TYPE ST_FastDoorStates :
STRUCT
	eState		: E_FastDoorState; //State
	eLastState	: E_FastDoorState; //Last state
END_STRUCT
END_TYPE

(* stored: Version 1.1.0.1, ProductVersion 3.1.4024.9
   DUT ST_FastDoorStates: Id {4c93962d-641b-476f-b7dc-0d33a715da0e} *)
